FUNCTION_BLOCK fb_LocalTime
VAR_INPUT

END_VAR
VAR_OUTPUT
  sLocalTime  : STRING;
  dtLocalTime : DT;
END_VAR
VAR
  //GetSysTime    : FW_GetSystemTime;
  //strFileTime   : T_FILETIME;
  strFileTime   : Tc2_Utilities.T_FILETIME64;
END_VAR

//GetSysTime(dwTimeLo=> strFileTime.dwLowDateTime, dwTimeHi=> strFileTime.dwHighDateTime);
strFileTime    := F_GetSystemTime();

sLocalTime  := SYSTEMTIME_TO_STRING( FILETIME64_TO_SYSTEMTIME( strFileTime ) );
dtLocalTime := systemtime_to_dt( FILETIME64_TO_SYSTEMTIME( strFileTime ) );

END_FUNCTION_BLOCK

(* stored: Version 1.1.0.1, ProductVersion 3.1.4026.13
   POU fb_LocalTime: Id {5bc42e5b-644f-451c-ae54-fd9900177cfc}, SpecialFunc None *)
